(* Logix 5000 project; controller BTS01 vendor 1 type 14 code 217 rev 32.14; software revision 32.04; part 7 of 15 *)
(* tags used below, declared in another part *)
   Alarm_Active : DINT;
   Alarm_TMR : TIMER[17,32];
   ALM_ENABLE : DINT[25];
   HMI_Global_Alarm_Ack_PB : BOOL;
   HMIAlarms : DINT[25];   // Alarm Trigger Array
   HMIAlarmsMsg : STRING64[17,32];   // Alarm Descriptions to Match Alarm Trigger Array
(* Alarm, continued *)

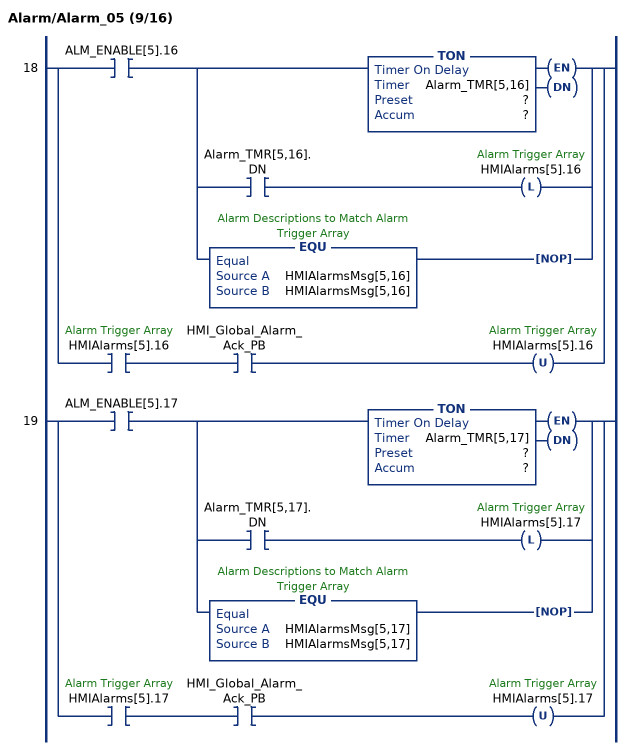
   [picture p111: Alarm/Alarm_05 rungs 18-19]
   18: [XIC(ALM_ENABLE[5].16) [TON(Alarm_TMR[5,16],?,?) ,XIC(Alarm_TMR[5,16].DN) OTL(HMIAlarms[5].16) ,EQU(HMIAlarmsMsg[5,16],HMIAlarmsMsg[5,16]) NOP() ] ,XIC(HMIAlarms[5].16) XIC(HMI_Global_Alarm_Ack_PB) OTU(HMIAlarms[5].16) ];
   19: [XIC(ALM_ENABLE[5].17) [TON(Alarm_TMR[5,17],?,?) ,XIC(Alarm_TMR[5,17].DN) OTL(HMIAlarms[5].17) ,EQU(HMIAlarmsMsg[5,17],HMIAlarmsMsg[5,17]) NOP() ] ,XIC(HMIAlarms[5].17) XIC(HMI_Global_Alarm_Ack_PB) OTU(HMIAlarms[5].17) ];
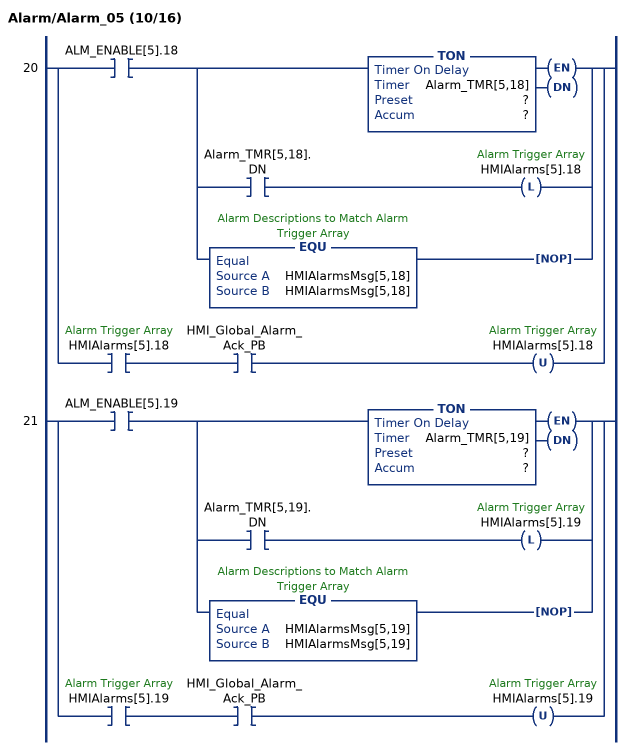
   20: [XIC(ALM_ENABLE[5].18) [TON(Alarm_TMR[5,18],?,?) ,XIC(Alarm_TMR[5,18].DN) OTL(HMIAlarms[5].18) ,EQU(HMIAlarmsMsg[5,18],HMIAlarmsMsg[5,18]) NOP() ] ,XIC(HMIAlarms[5].18) XIC(HMI_Global_Alarm_Ack_PB) OTU(HMIAlarms[5].18) ];
   21: [XIC(ALM_ENABLE[5].19) [TON(Alarm_TMR[5,19],?,?) ,XIC(Alarm_TMR[5,19].DN) OTL(HMIAlarms[5].19) ,EQU(HMIAlarmsMsg[5,19],HMIAlarmsMsg[5,19]) NOP() ] ,XIC(HMIAlarms[5].19) XIC(HMI_Global_Alarm_Ack_PB) OTU(HMIAlarms[5].19) ];
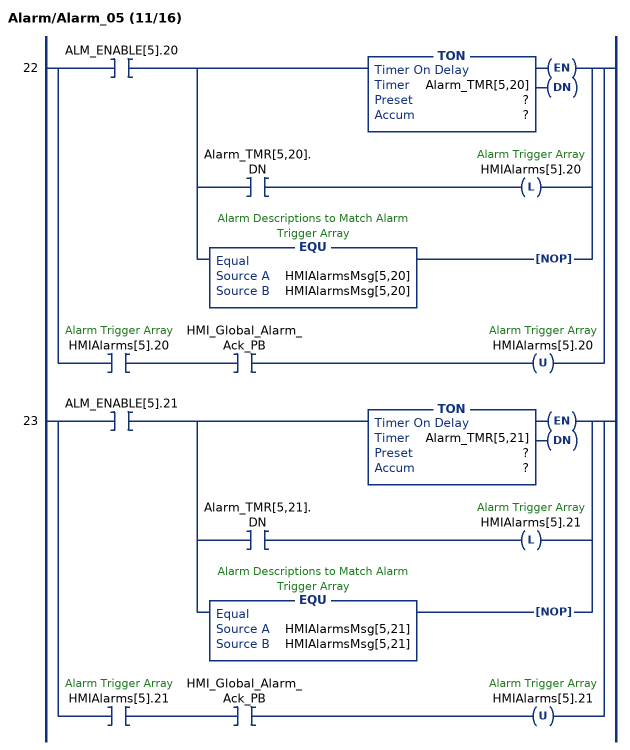
   22: [XIC(ALM_ENABLE[5].20) [TON(Alarm_TMR[5,20],?,?) ,XIC(Alarm_TMR[5,20].DN) OTL(HMIAlarms[5].20) ,EQU(HMIAlarmsMsg[5,20],HMIAlarmsMsg[5,20]) NOP() ] ,XIC(HMIAlarms[5].20) XIC(HMI_Global_Alarm_Ack_PB) OTU(HMIAlarms[5].20) ];
   23: [XIC(ALM_ENABLE[5].21) [TON(Alarm_TMR[5,21],?,?) ,XIC(Alarm_TMR[5,21].DN) OTL(HMIAlarms[5].21) ,EQU(HMIAlarmsMsg[5,21],HMIAlarmsMsg[5,21]) NOP() ] ,XIC(HMIAlarms[5].21) XIC(HMI_Global_Alarm_Ack_PB) OTU(HMIAlarms[5].21) ];
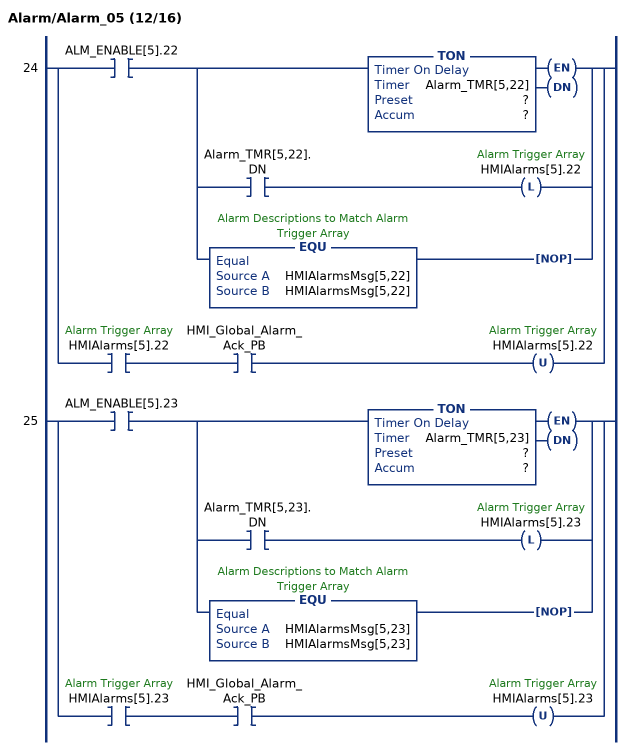
   24: [XIC(ALM_ENABLE[5].22) [TON(Alarm_TMR[5,22],?,?) ,XIC(Alarm_TMR[5,22].DN) OTL(HMIAlarms[5].22) ,EQU(HMIAlarmsMsg[5,22],HMIAlarmsMsg[5,22]) NOP() ] ,XIC(HMIAlarms[5].22) XIC(HMI_Global_Alarm_Ack_PB) OTU(HMIAlarms[5].22) ];
   25: [XIC(ALM_ENABLE[5].23) [TON(Alarm_TMR[5,23],?,?) ,XIC(Alarm_TMR[5,23].DN) OTL(HMIAlarms[5].23) ,EQU(HMIAlarmsMsg[5,23],HMIAlarmsMsg[5,23]) NOP() ] ,XIC(HMIAlarms[5].23) XIC(HMI_Global_Alarm_Ack_PB) OTU(HMIAlarms[5].23) ];
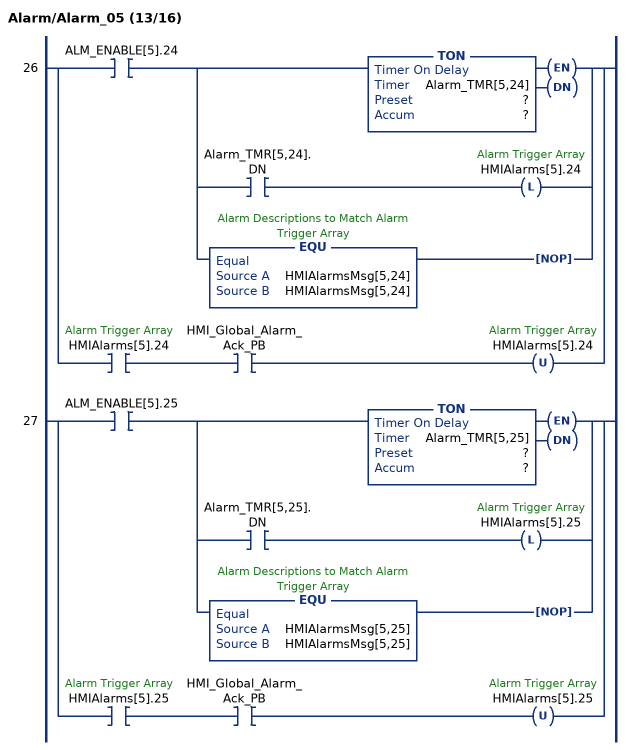
   26: [XIC(ALM_ENABLE[5].24) [TON(Alarm_TMR[5,24],?,?) ,XIC(Alarm_TMR[5,24].DN) OTL(HMIAlarms[5].24) ,EQU(HMIAlarmsMsg[5,24],HMIAlarmsMsg[5,24]) NOP() ] ,XIC(HMIAlarms[5].24) XIC(HMI_Global_Alarm_Ack_PB) OTU(HMIAlarms[5].24) ];
   27: [XIC(ALM_ENABLE[5].25) [TON(Alarm_TMR[5,25],?,?) ,XIC(Alarm_TMR[5,25].DN) OTL(HMIAlarms[5].25) ,EQU(HMIAlarmsMsg[5,25],HMIAlarmsMsg[5,25]) NOP() ] ,XIC(HMIAlarms[5].25) XIC(HMI_Global_Alarm_Ack_PB) OTU(HMIAlarms[5].25) ];
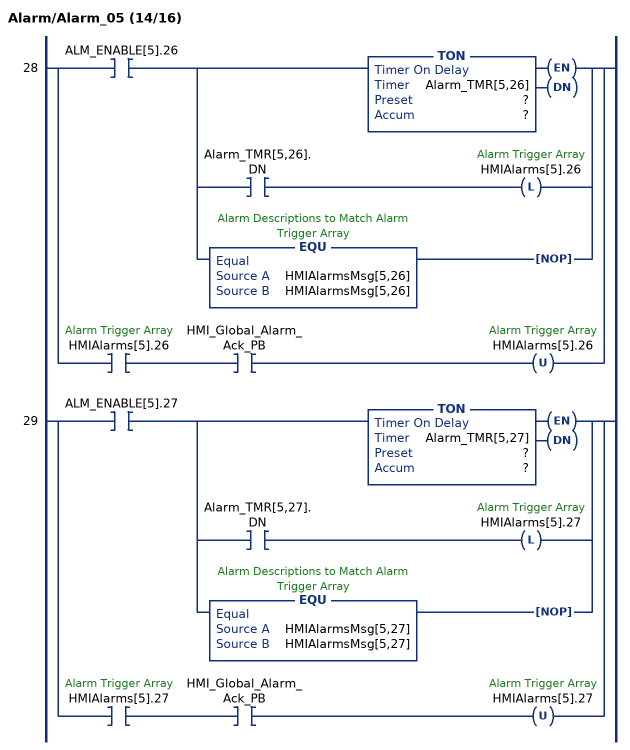
   28: [XIC(ALM_ENABLE[5].26) [TON(Alarm_TMR[5,26],?,?) ,XIC(Alarm_TMR[5,26].DN) OTL(HMIAlarms[5].26) ,EQU(HMIAlarmsMsg[5,26],HMIAlarmsMsg[5,26]) NOP() ] ,XIC(HMIAlarms[5].26) XIC(HMI_Global_Alarm_Ack_PB) OTU(HMIAlarms[5].26) ];
   29: [XIC(ALM_ENABLE[5].27) [TON(Alarm_TMR[5,27],?,?) ,XIC(Alarm_TMR[5,27].DN) OTL(HMIAlarms[5].27) ,EQU(HMIAlarmsMsg[5,27],HMIAlarmsMsg[5,27]) NOP() ] ,XIC(HMIAlarms[5].27) XIC(HMI_Global_Alarm_Ack_PB) OTU(HMIAlarms[5].27) ];
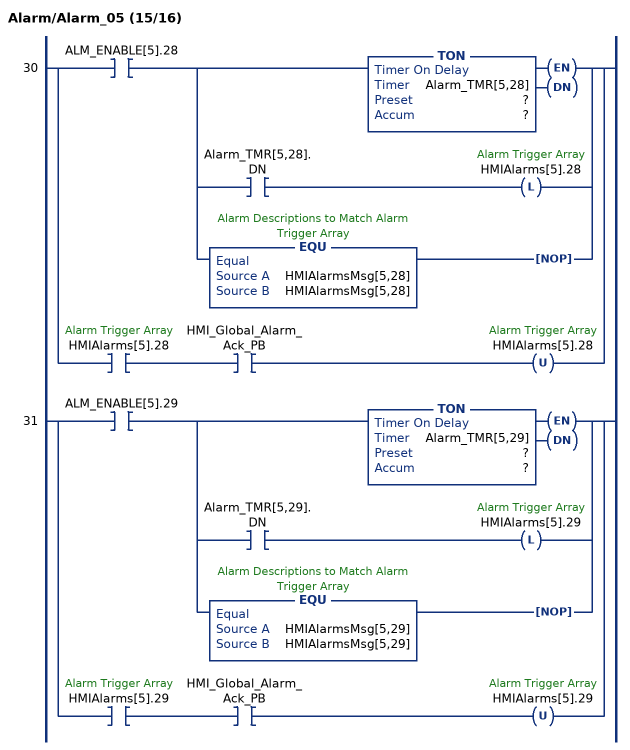
   30: [XIC(ALM_ENABLE[5].28) [TON(Alarm_TMR[5,28],?,?) ,XIC(Alarm_TMR[5,28].DN) OTL(HMIAlarms[5].28) ,EQU(HMIAlarmsMsg[5,28],HMIAlarmsMsg[5,28]) NOP() ] ,XIC(HMIAlarms[5].28) XIC(HMI_Global_Alarm_Ack_PB) OTU(HMIAlarms[5].28) ];
   31: [XIC(ALM_ENABLE[5].29) [TON(Alarm_TMR[5,29],?,?) ,XIC(Alarm_TMR[5,29].DN) OTL(HMIAlarms[5].29) ,EQU(HMIAlarmsMsg[5,29],HMIAlarmsMsg[5,29]) NOP() ] ,XIC(HMIAlarms[5].29) XIC(HMI_Global_Alarm_Ack_PB) OTU(HMIAlarms[5].29) ];
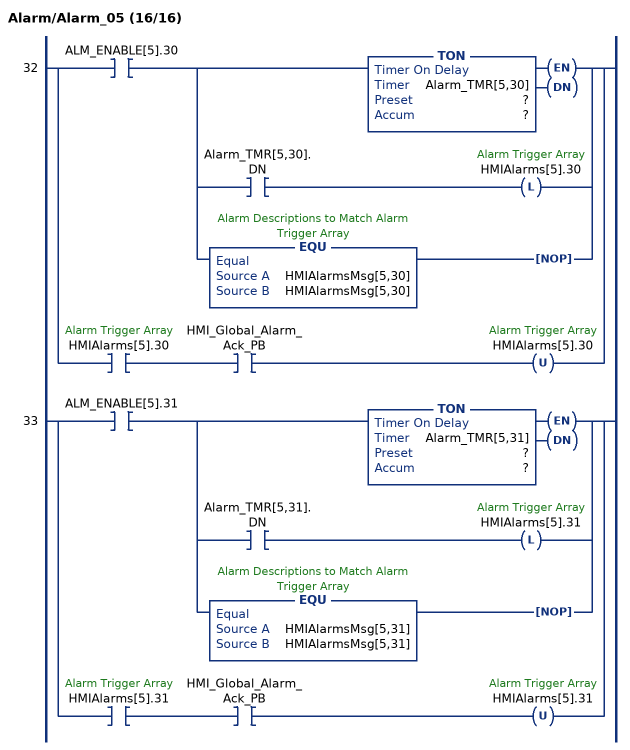
   32: [XIC(ALM_ENABLE[5].30) [TON(Alarm_TMR[5,30],?,?) ,XIC(Alarm_TMR[5,30].DN) OTL(HMIAlarms[5].30) ,EQU(HMIAlarmsMsg[5,30],HMIAlarmsMsg[5,30]) NOP() ] ,XIC(HMIAlarms[5].30) XIC(HMI_Global_Alarm_Ack_PB) OTU(HMIAlarms[5].30) ];
   33: [XIC(ALM_ENABLE[5].31) [TON(Alarm_TMR[5,31],?,?) ,XIC(Alarm_TMR[5,31].DN) OTL(HMIAlarms[5].31) ,EQU(HMIAlarmsMsg[5,31],HMIAlarmsMsg[5,31]) NOP() ] ,XIC(HMIAlarms[5].31) XIC(HMI_Global_Alarm_Ack_PB) OTU(HMIAlarms[5].31) ];
END_ROUTINE

ROUTINE Alarm_06   (* ladder *)
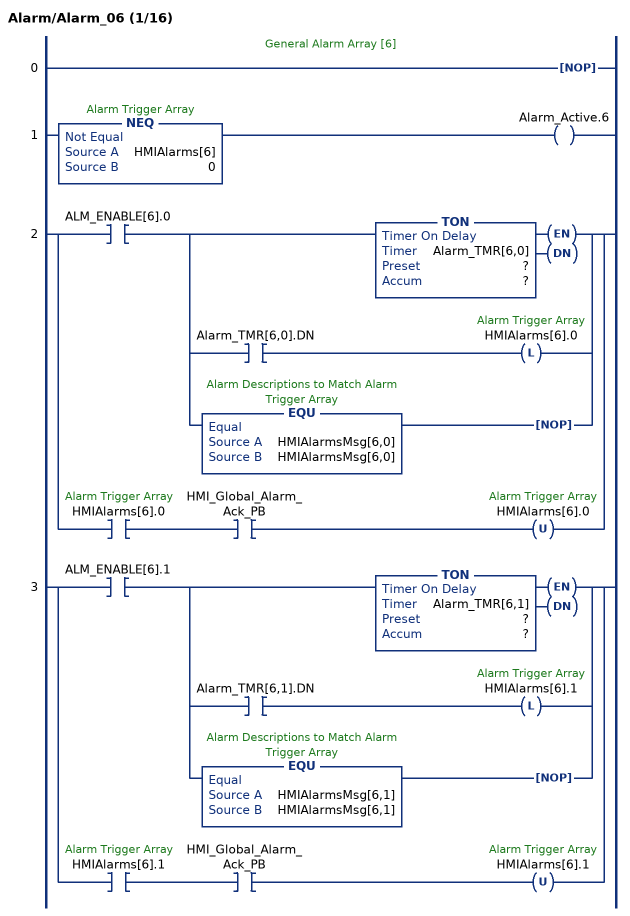
   // General Alarm Array [6]
   0: NOP();
   1: NEQ(HMIAlarms[6],0)OTE(Alarm_Active.6);
   2: [XIC(ALM_ENABLE[6].0) [TON(Alarm_TMR[6,0],?,?) ,XIC(Alarm_TMR[6,0].DN) OTL(HMIAlarms[6].0) ,EQU(HMIAlarmsMsg[6,0],HMIAlarmsMsg[6,0]) NOP() ] ,XIC(HMIAlarms[6].0) XIC(HMI_Global_Alarm_Ack_PB) OTU(HMIAlarms[6].0) ];
   3: [XIC(ALM_ENABLE[6].1) [TON(Alarm_TMR[6,1],?,?) ,XIC(Alarm_TMR[6,1].DN) OTL(HMIAlarms[6].1) ,EQU(HMIAlarmsMsg[6,1],HMIAlarmsMsg[6,1]) NOP() ] ,XIC(HMIAlarms[6].1) XIC(HMI_Global_Alarm_Ack_PB) OTU(HMIAlarms[6].1) ];
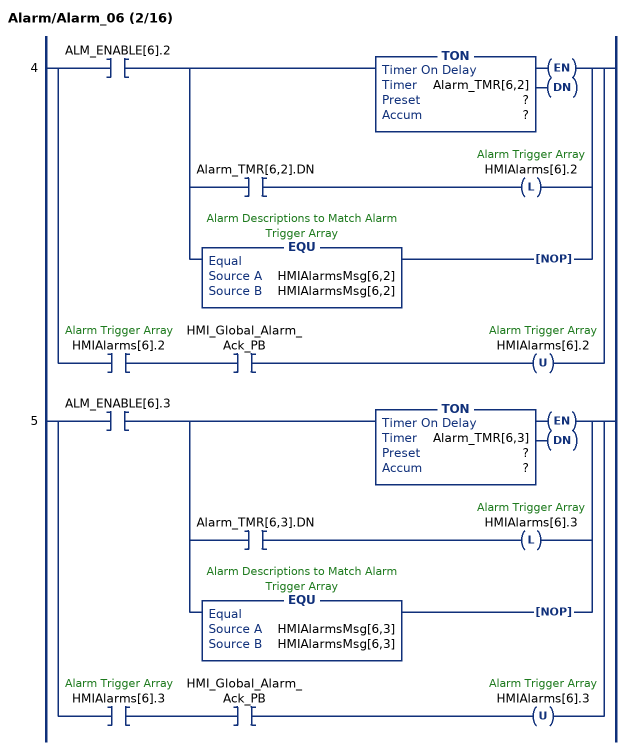
   4: [XIC(ALM_ENABLE[6].2) [TON(Alarm_TMR[6,2],?,?) ,XIC(Alarm_TMR[6,2].DN) OTL(HMIAlarms[6].2) ,EQU(HMIAlarmsMsg[6,2],HMIAlarmsMsg[6,2]) NOP() ] ,XIC(HMIAlarms[6].2) XIC(HMI_Global_Alarm_Ack_PB) OTU(HMIAlarms[6].2) ];
   5: [XIC(ALM_ENABLE[6].3) [TON(Alarm_TMR[6,3],?,?) ,XIC(Alarm_TMR[6,3].DN) OTL(HMIAlarms[6].3) ,EQU(HMIAlarmsMsg[6,3],HMIAlarmsMsg[6,3]) NOP() ] ,XIC(HMIAlarms[6].3) XIC(HMI_Global_Alarm_Ack_PB) OTU(HMIAlarms[6].3) ];
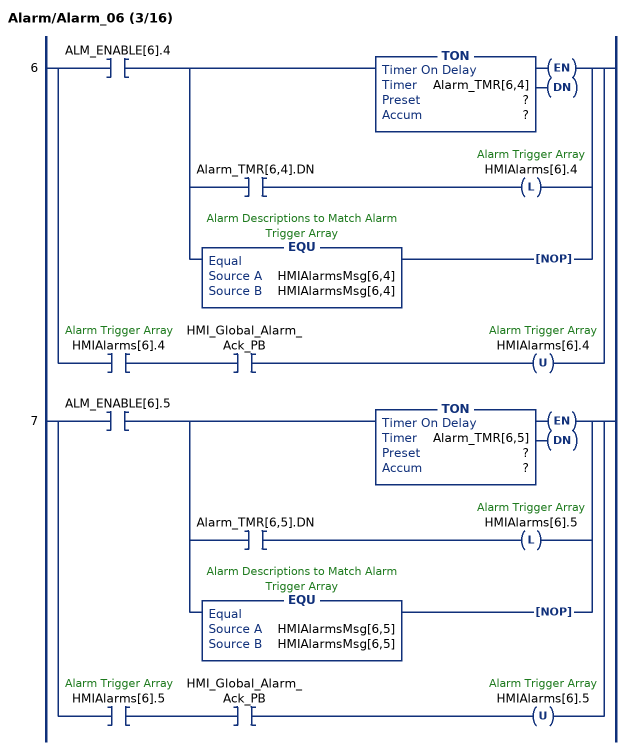
   6: [XIC(ALM_ENABLE[6].4) [TON(Alarm_TMR[6,4],?,?) ,XIC(Alarm_TMR[6,4].DN) OTL(HMIAlarms[6].4) ,EQU(HMIAlarmsMsg[6,4],HMIAlarmsMsg[6,4]) NOP() ] ,XIC(HMIAlarms[6].4) XIC(HMI_Global_Alarm_Ack_PB) OTU(HMIAlarms[6].4) ];
   7: [XIC(ALM_ENABLE[6].5) [TON(Alarm_TMR[6,5],?,?) ,XIC(Alarm_TMR[6,5].DN) OTL(HMIAlarms[6].5) ,EQU(HMIAlarmsMsg[6,5],HMIAlarmsMsg[6,5]) NOP() ] ,XIC(HMIAlarms[6].5) XIC(HMI_Global_Alarm_Ack_PB) OTU(HMIAlarms[6].5) ];
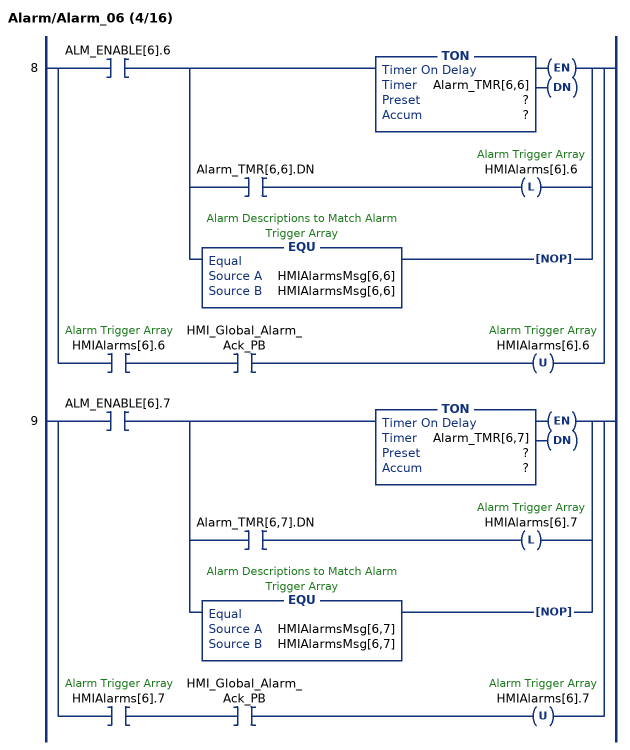
   8: [XIC(ALM_ENABLE[6].6) [TON(Alarm_TMR[6,6],?,?) ,XIC(Alarm_TMR[6,6].DN) OTL(HMIAlarms[6].6) ,EQU(HMIAlarmsMsg[6,6],HMIAlarmsMsg[6,6]) NOP() ] ,XIC(HMIAlarms[6].6) XIC(HMI_Global_Alarm_Ack_PB) OTU(HMIAlarms[6].6) ];
   9: [XIC(ALM_ENABLE[6].7) [TON(Alarm_TMR[6,7],?,?) ,XIC(Alarm_TMR[6,7].DN) OTL(HMIAlarms[6].7) ,EQU(HMIAlarmsMsg[6,7],HMIAlarmsMsg[6,7]) NOP() ] ,XIC(HMIAlarms[6].7) XIC(HMI_Global_Alarm_Ack_PB) OTU(HMIAlarms[6].7) ];
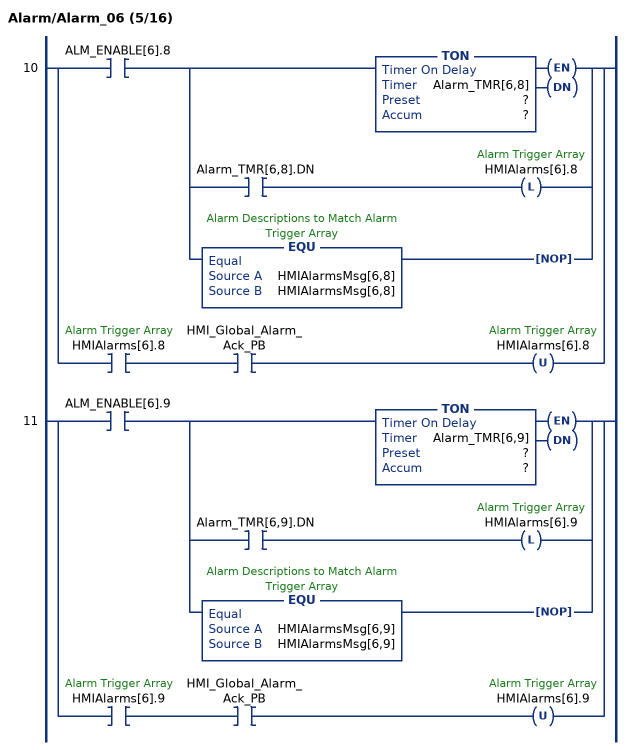
   10: [XIC(ALM_ENABLE[6].8) [TON(Alarm_TMR[6,8],?,?) ,XIC(Alarm_TMR[6,8].DN) OTL(HMIAlarms[6].8) ,EQU(HMIAlarmsMsg[6,8],HMIAlarmsMsg[6,8]) NOP() ] ,XIC(HMIAlarms[6].8) XIC(HMI_Global_Alarm_Ack_PB) OTU(HMIAlarms[6].8) ];
   11: [XIC(ALM_ENABLE[6].9) [TON(Alarm_TMR[6,9],?,?) ,XIC(Alarm_TMR[6,9].DN) OTL(HMIAlarms[6].9) ,EQU(HMIAlarmsMsg[6,9],HMIAlarmsMsg[6,9]) NOP() ] ,XIC(HMIAlarms[6].9) XIC(HMI_Global_Alarm_Ack_PB) OTU(HMIAlarms[6].9) ];
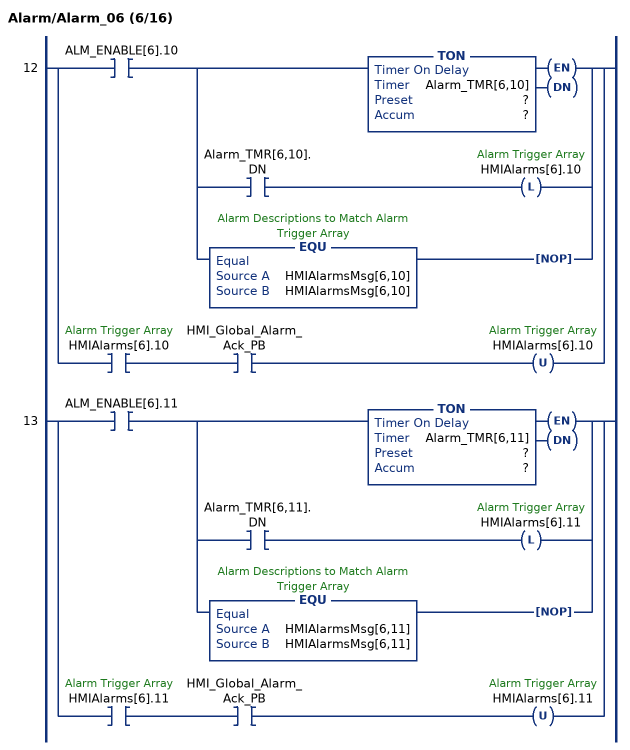
   12: [XIC(ALM_ENABLE[6].10) [TON(Alarm_TMR[6,10],?,?) ,XIC(Alarm_TMR[6,10].DN) OTL(HMIAlarms[6].10) ,EQU(HMIAlarmsMsg[6,10],HMIAlarmsMsg[6,10]) NOP() ] ,XIC(HMIAlarms[6].10) XIC(HMI_Global_Alarm_Ack_PB) OTU(HMIAlarms[6].10) ];
   13: [XIC(ALM_ENABLE[6].11) [TON(Alarm_TMR[6,11],?,?) ,XIC(Alarm_TMR[6,11].DN) OTL(HMIAlarms[6].11) ,EQU(HMIAlarmsMsg[6,11],HMIAlarmsMsg[6,11]) NOP() ] ,XIC(HMIAlarms[6].11) XIC(HMI_Global_Alarm_Ack_PB) OTU(HMIAlarms[6].11) ];
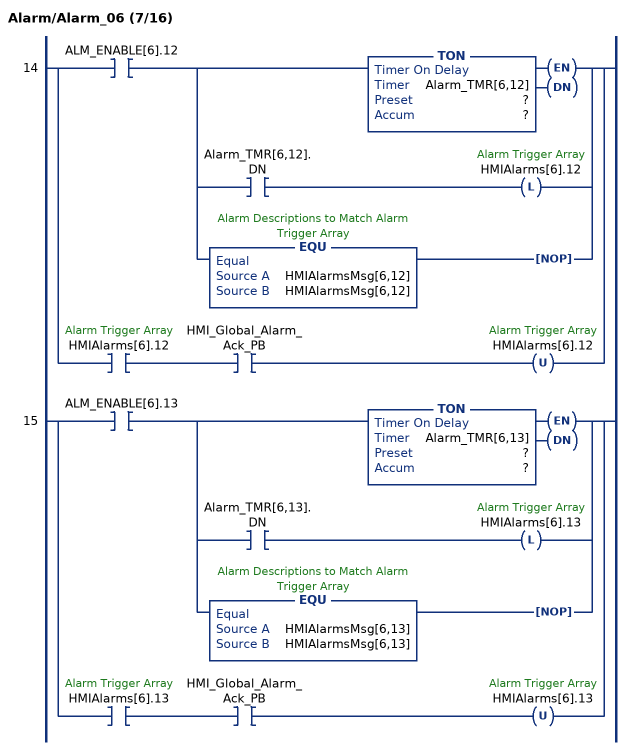
   14: [XIC(ALM_ENABLE[6].12) [TON(Alarm_TMR[6,12],?,?) ,XIC(Alarm_TMR[6,12].DN) OTL(HMIAlarms[6].12) ,EQU(HMIAlarmsMsg[6,12],HMIAlarmsMsg[6,12]) NOP() ] ,XIC(HMIAlarms[6].12) XIC(HMI_Global_Alarm_Ack_PB) OTU(HMIAlarms[6].12) ];
   15: [XIC(ALM_ENABLE[6].13) [TON(Alarm_TMR[6,13],?,?) ,XIC(Alarm_TMR[6,13].DN) OTL(HMIAlarms[6].13) ,EQU(HMIAlarmsMsg[6,13],HMIAlarmsMsg[6,13]) NOP() ] ,XIC(HMIAlarms[6].13) XIC(HMI_Global_Alarm_Ack_PB) OTU(HMIAlarms[6].13) ];
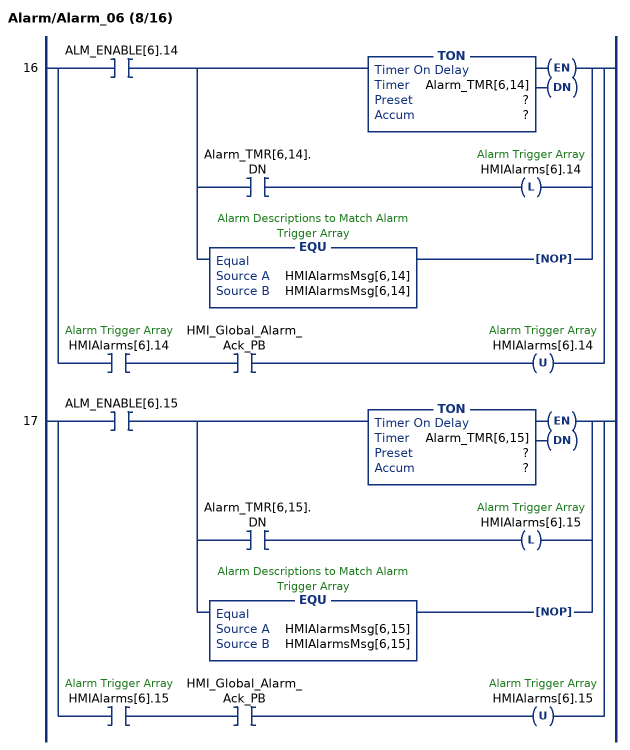
   16: [XIC(ALM_ENABLE[6].14) [TON(Alarm_TMR[6,14],?,?) ,XIC(Alarm_TMR[6,14].DN) OTL(HMIAlarms[6].14) ,EQU(HMIAlarmsMsg[6,14],HMIAlarmsMsg[6,14]) NOP() ] ,XIC(HMIAlarms[6].14) XIC(HMI_Global_Alarm_Ack_PB) OTU(HMIAlarms[6].14) ];
   17: [XIC(ALM_ENABLE[6].15) [TON(Alarm_TMR[6,15],?,?) ,XIC(Alarm_TMR[6,15].DN) OTL(HMIAlarms[6].15) ,EQU(HMIAlarmsMsg[6,15],HMIAlarmsMsg[6,15]) NOP() ] ,XIC(HMIAlarms[6].15) XIC(HMI_Global_Alarm_Ack_PB) OTU(HMIAlarms[6].15) ];
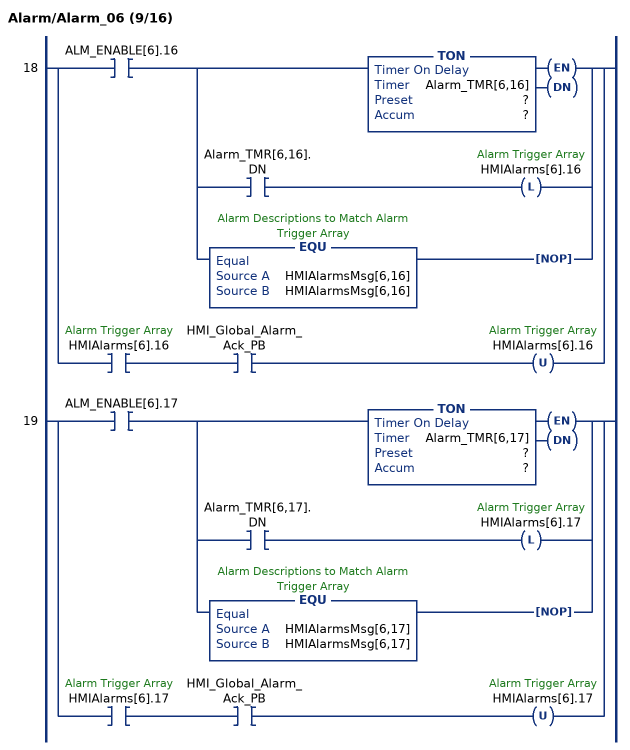
   18: [XIC(ALM_ENABLE[6].16) [TON(Alarm_TMR[6,16],?,?) ,XIC(Alarm_TMR[6,16].DN) OTL(HMIAlarms[6].16) ,EQU(HMIAlarmsMsg[6,16],HMIAlarmsMsg[6,16]) NOP() ] ,XIC(HMIAlarms[6].16) XIC(HMI_Global_Alarm_Ack_PB) OTU(HMIAlarms[6].16) ];
   19: [XIC(ALM_ENABLE[6].17) [TON(Alarm_TMR[6,17],?,?) ,XIC(Alarm_TMR[6,17].DN) OTL(HMIAlarms[6].17) ,EQU(HMIAlarmsMsg[6,17],HMIAlarmsMsg[6,17]) NOP() ] ,XIC(HMIAlarms[6].17) XIC(HMI_Global_Alarm_Ack_PB) OTU(HMIAlarms[6].17) ];
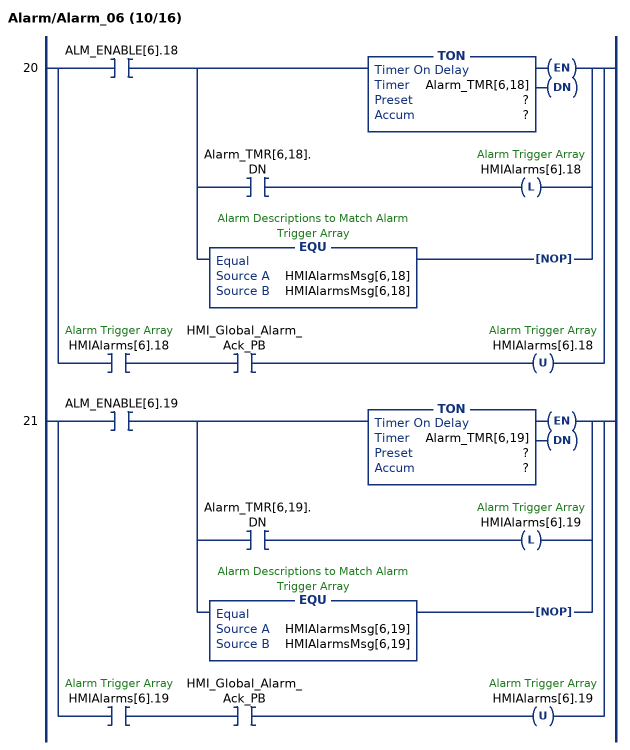
   20: [XIC(ALM_ENABLE[6].18) [TON(Alarm_TMR[6,18],?,?) ,XIC(Alarm_TMR[6,18].DN) OTL(HMIAlarms[6].18) ,EQU(HMIAlarmsMsg[6,18],HMIAlarmsMsg[6,18]) NOP() ] ,XIC(HMIAlarms[6].18) XIC(HMI_Global_Alarm_Ack_PB) OTU(HMIAlarms[6].18) ];
   21: [XIC(ALM_ENABLE[6].19) [TON(Alarm_TMR[6,19],?,?) ,XIC(Alarm_TMR[6,19].DN) OTL(HMIAlarms[6].19) ,EQU(HMIAlarmsMsg[6,19],HMIAlarmsMsg[6,19]) NOP() ] ,XIC(HMIAlarms[6].19) XIC(HMI_Global_Alarm_Ack_PB) OTU(HMIAlarms[6].19) ];
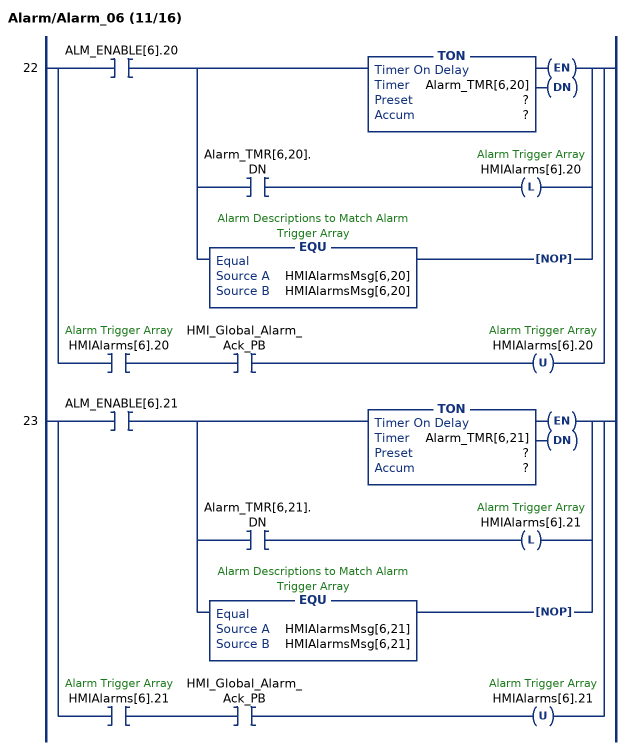
   22: [XIC(ALM_ENABLE[6].20) [TON(Alarm_TMR[6,20],?,?) ,XIC(Alarm_TMR[6,20].DN) OTL(HMIAlarms[6].20) ,EQU(HMIAlarmsMsg[6,20],HMIAlarmsMsg[6,20]) NOP() ] ,XIC(HMIAlarms[6].20) XIC(HMI_Global_Alarm_Ack_PB) OTU(HMIAlarms[6].20) ];
   23: [XIC(ALM_ENABLE[6].21) [TON(Alarm_TMR[6,21],?,?) ,XIC(Alarm_TMR[6,21].DN) OTL(HMIAlarms[6].21) ,EQU(HMIAlarmsMsg[6,21],HMIAlarmsMsg[6,21]) NOP() ] ,XIC(HMIAlarms[6].21) XIC(HMI_Global_Alarm_Ack_PB) OTU(HMIAlarms[6].21) ];
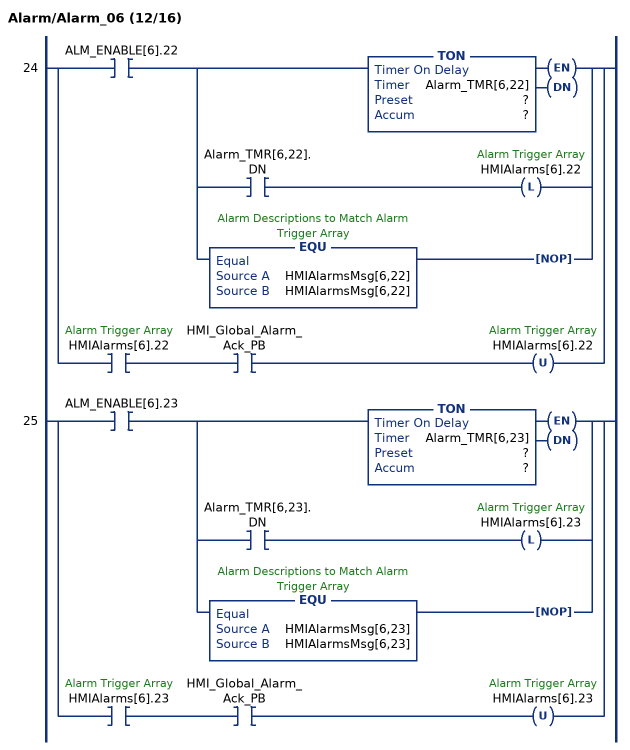
   24: [XIC(ALM_ENABLE[6].22) [TON(Alarm_TMR[6,22],?,?) ,XIC(Alarm_TMR[6,22].DN) OTL(HMIAlarms[6].22) ,EQU(HMIAlarmsMsg[6,22],HMIAlarmsMsg[6,22]) NOP() ] ,XIC(HMIAlarms[6].22) XIC(HMI_Global_Alarm_Ack_PB) OTU(HMIAlarms[6].22) ];
   25: [XIC(ALM_ENABLE[6].23) [TON(Alarm_TMR[6,23],?,?) ,XIC(Alarm_TMR[6,23].DN) OTL(HMIAlarms[6].23) ,EQU(HMIAlarmsMsg[6,23],HMIAlarmsMsg[6,23]) NOP() ] ,XIC(HMIAlarms[6].23) XIC(HMI_Global_Alarm_Ack_PB) OTU(HMIAlarms[6].23) ];
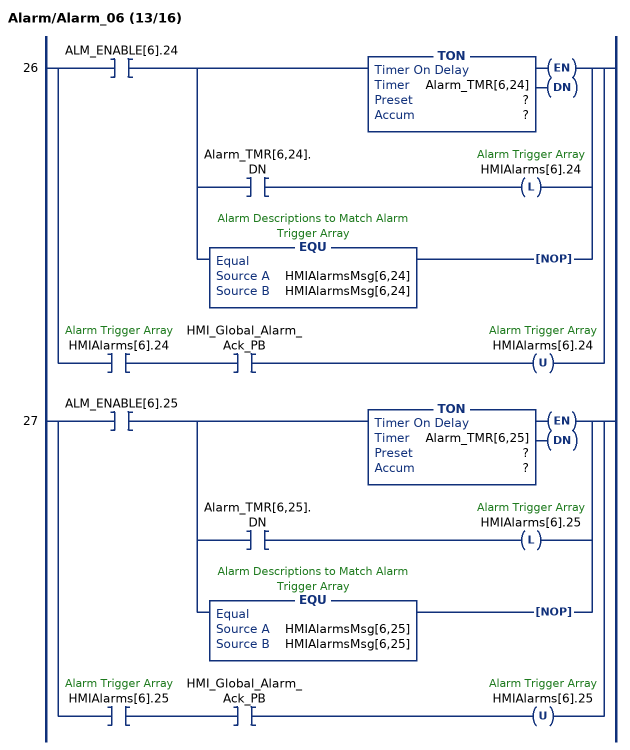
   26: [XIC(ALM_ENABLE[6].24) [TON(Alarm_TMR[6,24],?,?) ,XIC(Alarm_TMR[6,24].DN) OTL(HMIAlarms[6].24) ,EQU(HMIAlarmsMsg[6,24],HMIAlarmsMsg[6,24]) NOP() ] ,XIC(HMIAlarms[6].24) XIC(HMI_Global_Alarm_Ack_PB) OTU(HMIAlarms[6].24) ];
   27: [XIC(ALM_ENABLE[6].25) [TON(Alarm_TMR[6,25],?,?) ,XIC(Alarm_TMR[6,25].DN) OTL(HMIAlarms[6].25) ,EQU(HMIAlarmsMsg[6,25],HMIAlarmsMsg[6,25]) NOP() ] ,XIC(HMIAlarms[6].25) XIC(HMI_Global_Alarm_Ack_PB) OTU(HMIAlarms[6].25) ];
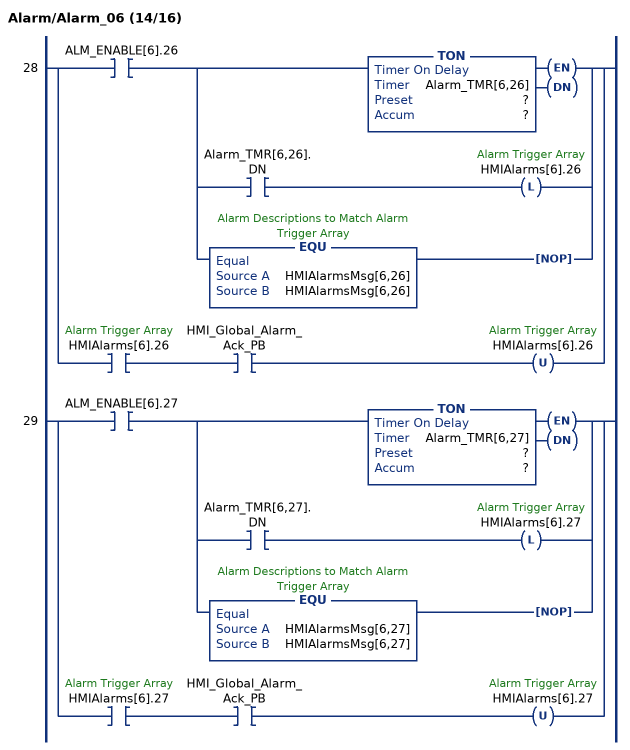
   28: [XIC(ALM_ENABLE[6].26) [TON(Alarm_TMR[6,26],?,?) ,XIC(Alarm_TMR[6,26].DN) OTL(HMIAlarms[6].26) ,EQU(HMIAlarmsMsg[6,26],HMIAlarmsMsg[6,26]) NOP() ] ,XIC(HMIAlarms[6].26) XIC(HMI_Global_Alarm_Ack_PB) OTU(HMIAlarms[6].26) ];
   29: [XIC(ALM_ENABLE[6].27) [TON(Alarm_TMR[6,27],?,?) ,XIC(Alarm_TMR[6,27].DN) OTL(HMIAlarms[6].27) ,EQU(HMIAlarmsMsg[6,27],HMIAlarmsMsg[6,27]) NOP() ] ,XIC(HMIAlarms[6].27) XIC(HMI_Global_Alarm_Ack_PB) OTU(HMIAlarms[6].27) ];
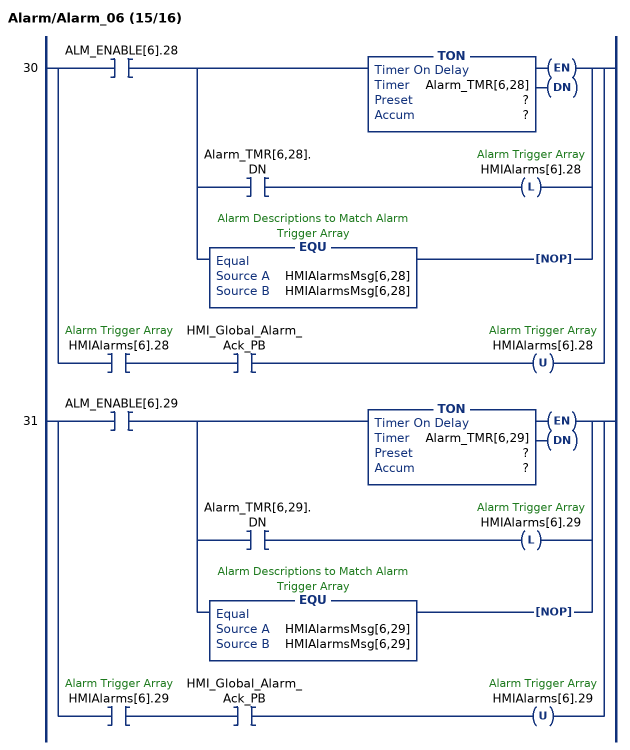
   30: [XIC(ALM_ENABLE[6].28) [TON(Alarm_TMR[6,28],?,?) ,XIC(Alarm_TMR[6,28].DN) OTL(HMIAlarms[6].28) ,EQU(HMIAlarmsMsg[6,28],HMIAlarmsMsg[6,28]) NOP() ] ,XIC(HMIAlarms[6].28) XIC(HMI_Global_Alarm_Ack_PB) OTU(HMIAlarms[6].28) ];
   31: [XIC(ALM_ENABLE[6].29) [TON(Alarm_TMR[6,29],?,?) ,XIC(Alarm_TMR[6,29].DN) OTL(HMIAlarms[6].29) ,EQU(HMIAlarmsMsg[6,29],HMIAlarmsMsg[6,29]) NOP() ] ,XIC(HMIAlarms[6].29) XIC(HMI_Global_Alarm_Ack_PB) OTU(HMIAlarms[6].29) ];
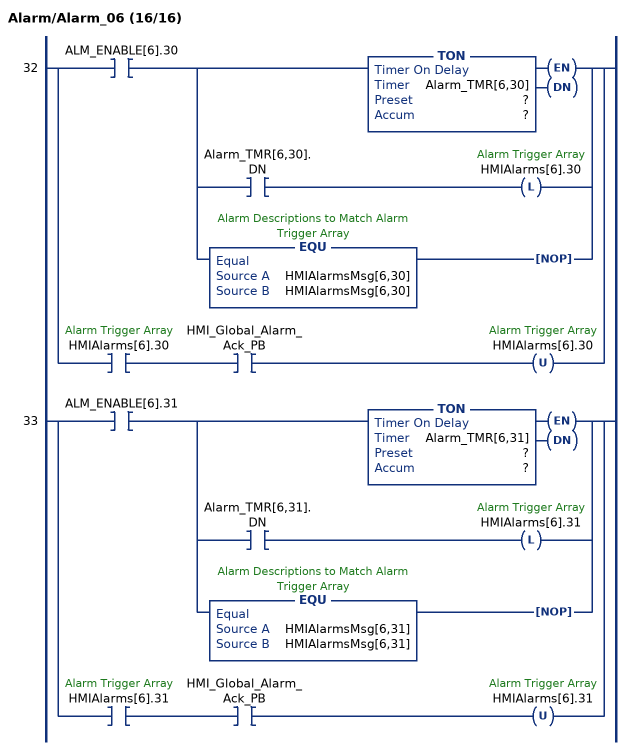
   32: [XIC(ALM_ENABLE[6].30) [TON(Alarm_TMR[6,30],?,?) ,XIC(Alarm_TMR[6,30].DN) OTL(HMIAlarms[6].30) ,EQU(HMIAlarmsMsg[6,30],HMIAlarmsMsg[6,30]) NOP() ] ,XIC(HMIAlarms[6].30) XIC(HMI_Global_Alarm_Ack_PB) OTU(HMIAlarms[6].30) ];
   33: [XIC(ALM_ENABLE[6].31) [TON(Alarm_TMR[6,31],?,?) ,XIC(Alarm_TMR[6,31].DN) OTL(HMIAlarms[6].31) ,EQU(HMIAlarmsMsg[6,31],HMIAlarmsMsg[6,31]) NOP() ] ,XIC(HMIAlarms[6].31) XIC(HMI_Global_Alarm_Ack_PB) OTU(HMIAlarms[6].31) ];
END_ROUTINE
